# EPICS substitutions: EX2/scr/neurons.substitutions
file network.template {
	pattern { name, name-next, in1, w1, in2, w2, in3, w3, in4, w4}

		{ "11", "12-sum", "01", "01-11", "11", "11-11", "12", "12-11", "13", "13-11" }
		{ "12", "13-sum", "01", "01-12", "11", "11-12", "12", "12-12", "13", "13-12" }
		{ "13", "11-ac", "01", "01-13", "11", "11-13", "12", "12-13", "13", "13-13" }

		{ "21", "22-sum", "11", "11-21", "12", "12-21", "13", "13-21", "null", "null" }
		{ "22", "23-sum", "11", "11-22", "12", "12-22", "13", "13-22", "null", "null" }
		{ "23", "21-ac", "11", "11-23", "12", "12-23", "13", "13-23", "null", "null" }
}

file ac.template {
	pattern { name, name-next }
		{ "11", "12-ac" }
		{ "12", "13-ac" }
		{ "13", "21-sum" }

		{ "21", "22-ac" }
		{ "22", "23-ac" }
		{ "23", "score-fanout" }
}

file softmax.template {
	pattern { name, other1, other2 }
		{ "21", "22", "23" }
		{ "22", "21", "23" }
		{ "23", "21", "22" }
}

file weights.template {
	pattern { name1, name2, weight }
		{ "01", "11", "2.610053" }
		{ "01", "12", "4.688208" }
		{ "01", "13", "-15.884566" }

		{ "11", "11", "-1.229400" }
		{ "12", "11", "0.389088" }
		{ "13", "11", "0.111757" }

		{ "11", "12", "-10.916350" }
		{ "12", "12", "3.052341" }
		{ "13", "12", "0.845389" }

		{ "11", "13", "28.358418" }
		{ "12", "13", "-7.38725" }
		{ "13", "13", "-1.968287" }

		{ "11", "21", "5.493579" }
		{ "12", "21", "18.733213" }
		{ "13", "21", "-35.217319" }

		{ "11", "22", "1.113441" }
		{ "12", "22", "-0.137917" }
		{ "13", "22", "1.186039" }

		{ "11", "23", "-7.128529" }
		{ "12", "23", "-23.056977" }
		{ "13", "23", "34.451607" }
}

file bias.template {
	pattern { name, bias }

		{ "11", "-0.993523" }
		{ "12", "1.122133" }
		{ "13", "-1.157693" }

		{ "21", "2.195953" }
		{ "22", "1.146973" }
		{ "23", "-4.095017" }
}
